PROGRAM _4000_PRG_Pausing
VAR_IN_OUT
    CurrentStep : ActiveStep;
    NextStep    : DINT;
END_VAR
VAR_INPUT
    StepTimerSeconds   : DINT;
    RetrySignal        : BOOL;
    StateMachineStatus : ST_SM_Status;
END_VAR
VAR
    fbStep4000 : FB_SequenceStep; // Pausing prepare
    fbStep4002 : FB_SequenceStep; // Pausing execute
    step4000Perms : INT := -1;
    step4002Perms : INT := -1;
END_VAR


// STEP 4000 - PAUSING PREPARE
fbStep4000(
    inpStep := CurrentStep.Step,
    cfgStep := 4000,
    cfgNextStep := 4002,
    inpStepTimerSeconds := StepTimerSeconds,
    inpRetry := RetrySignal,
    inpStepPermissives := step4000Perms,
    cfgStepTimeout := 5,
    inpFaultStep := FALSE,
    ActiveStep := CurrentStep
);
IF fbStep4000.outStepActive THEN
    IF fbStep4000.outNextStep = fbStep4000.cfgStep THEN
        IF StepTimerSeconds < 2 THEN
            step4000Perms := 16#FFFE;
        ELSE
            step4000Perms := -1;
        END_IF;
    END_IF;
    CurrentStep.PermsHMI.Name := 'Pausing Prepare';
    CurrentStep.PermsHMI.Desc[0] := 'Prepare to Pause';
    CurrentStep.PermsHMI.Desc[1] := 'Buffer Operations';
    CurrentStep.PermsHMI.Desc[2] := 'Safe To Pause';
    NextStep := fbStep4000.outNextStep;
ELSE
    step4000Perms := 16#FFFE;
END_IF;

// STEP 4002 - PAUSING EXECUTE
fbStep4002(
    inpStep := CurrentStep.Step,
    cfgStep := 4002,
    cfgNextStep := 0, // sequence complete
    inpStepTimerSeconds := StepTimerSeconds,
    inpRetry := RetrySignal,
    inpStepPermissives := step4002Perms,
    cfgStepTimeout := 8,
    inpFaultStep := FALSE,
    ActiveStep := CurrentStep
);
IF fbStep4002.outStepActive THEN
    IF fbStep4002.outNextStep = fbStep4002.cfgStep THEN
        IF StepTimerSeconds < 5 THEN
            step4002Perms := 16#FFFD;
        ELSE
            step4002Perms := -1;
        END_IF;
    END_IF;
    CurrentStep.PermsHMI.Name := 'Pausing Execute';
    CurrentStep.PermsHMI.Desc[0] := 'Pausing';
    CurrentStep.PermsHMI.Desc[1] := 'Drive/Actuator Hold';
    CurrentStep.PermsHMI.Desc[2] := 'Safe State';
    NextStep := fbStep4002.outNextStep;
ELSE
    step4002Perms := 16#FFFD;
END_IF;

END_PROGRAM

(* stored: Version 1.1.0.1, ProductVersion 3.1.4024.13
   POU _4000_PRG_Pausing: Id {8e2c6c3f-6f2a-4c03-bb33-4ec0b5f1b4d0}, SpecialFunc None *)
